/// This is the error type used in this library.
TYPE Error :
STRUCT
	Active : BOOL; // `TRUE` signals an active error
	Code : INT; // Error code of type `ErrorCodes`
	Info : Tc2_System.T_MaxString; // Plain text error message
END_STRUCT
END_TYPE

(* stored: Version 1.1.0.1
   DUT Error: Id {23c996c0-f051-4322-bcdc-8cc9475229f8} *)
